// TIA Portal V17 export
// export: Created 2024-08-20T13:26:11.9403241Z, ExportSetting WithDefaults, DisplayName Totally Integrated Automation Portal, DisplayVersion V17 Update 4, DisplayName TIA Portal Openness, DisplayVersion V17 Update 4, DisplayName TIA Portal Version Control Interface, DisplayVersion V17, DisplayName STEP 7 Professional, DisplayVersion V17 Update 4, DisplayName STEP 7 Safety, DisplayVersion V17, DisplayName WinCC Advanced, DisplayVersion V17 Update 4
DATA_BLOCK "LOOP_DB"   // DB3
VERSION : 0.1
// stored: AutoNumber true, DBAccessibleFromOPCUA true, InstanceOfName LOOP, InstanceOfType FB
"LOOP"
   // VAR
   //    PULSO : Bool;
   //    AuxLoop : Bool;
   //    N_L00P : Int;
   //    Aux_N_LOOP : Int;
   //    Loop : Int;
   // END_VAR
BEGIN
END_DATA_BLOCK
